/// General move parameter strucure
TYPE ST_AxisMoveParameter :
STRUCT
	fVelocity: LREAL;
	fAcceleration: LREAL;
	fDeceleration: LREAL;
	fJerk: LREAL;
	eBufferMode: MC_BufferMode := MC_Aborting;
	stOptions: ST_MoveOptions;
END_STRUCT
END_TYPE

(* stored: Version 1.1.0.1, ProductVersion 3.1.4022.9
   DUT ST_AxisMoveParameter: Id {216ee36e-d0e1-450d-84db-fe61ab4dd2db} *)
